FUNCTION_BLOCK FB_SlaveCountDiagnosis
VAR_IN_OUT
	eEtherCATMaster				:E_EtherCATMaster;	
END_VAR
VAR_OUTPUT
	bError						:BOOL;								//エラー発生を出力
END_VAR
VAR
	uiSlaveCount 		AT%I*	:UINT;								//PDデータとリンク
	uiCfgSlaveCount 	AT%I*	:UINT;								//PDデータとリンク
	
	sMasterName					:STRING;
	
	fbBitREdge					:R_TRIG;
	fbMessage					:FB_TcMessage;
	i							:INT;
END_VAR

//マスター名を入力
	IF sMasterName<>TO_STRING(eEtherCATMaster) THEN
		sMasterName:=TO_STRING(eEtherCATMaster);
	END_IF

//エラー状態を出力
	bError:=uiSlaveCount<>uiCfgSlaveCount OR uiSlaveCount=0 OR uiCfgSlaveCount=0;

//エラーをEventloggerへ
	fbBitREdge(CLK:=bError);
	
	IF fbBitREdge.Q THEN
		fbMessage.ipArguments.Clear().AddString(sMasterName);
		fbMessage.Send();
	END_IF

//FB_Init は常に暗黙的に使用可能で、主に初期化に使用されます。
//戻り値は評価されません。特定の結果を得るために、メソッドを明示的に宣言し、
//そのメソッドに標準の初期化コードをもったコードを追加することができます。戻り値を評価できます。
METHOD FB_Init: BOOL
VAR_INPUT
    bInitRetains: BOOL; // TRUE: 保持変数は初期化されます (ウォーム リセット、あるいはコールド リセット)
    bInCopyCode: BOOL;  // TRUE: 後でコードをコピーする (オンライン変更) ために、インスタンスをコピーします。
END_VAR
fbMessage.CreateEx(Tc_Events.TkEtherCATMasterDiagnosisEventClass.MismatchSlaveCountCfgSlaveCount);
END_METHOD

END_FUNCTION_BLOCK

(* stored: Version 1.1.0.1, ProductVersion 3.1.4026.18
   POU FB_SlaveCountDiagnosis: Id {02ab8264-55ea-46ed-995e-d44a3481583b}, SpecialFunc None
   Method FB_Init: Id {0370321f-7f5d-475b-838a-b30d147a8230} *)
